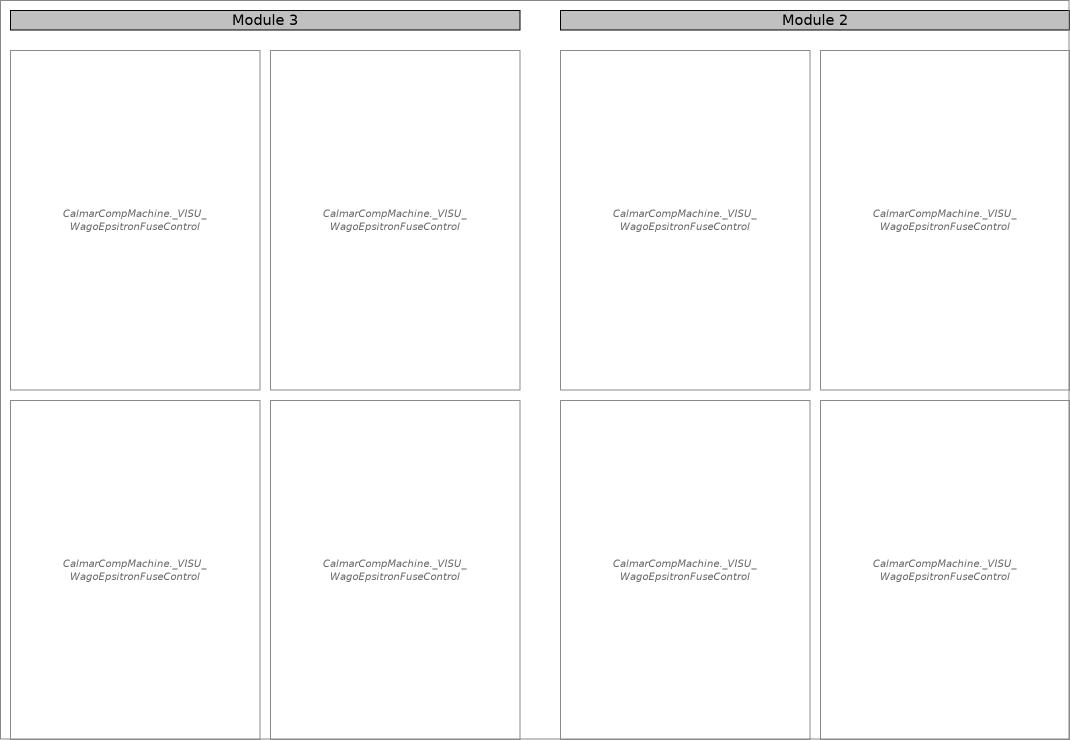
VISUALIZATION _VISU_FUSE_CONTROL  // 1070x740
VAR_IN_OUT
	mInst : FB_WeuPowerControl;
END_VAR
    Frame (820,50 250x340)
        shows CalmarCompMachine._VISU_WagoEpsitronFuseControl(m_Inst_Fb := PRG_MACHINE.fbPowerControl.fb_EpsitronFuseControlF70M1)
    Frame (560,50 250x340)
        shows CalmarCompMachine._VISU_WagoEpsitronFuseControl(m_Inst_Fb := PRG_MACHINE.fbPowerControl.fb_EpsitronFuseControlF90M1)
    Frame (270,50 250x340)
        shows CalmarCompMachine._VISU_WagoEpsitronFuseControl(m_Inst_Fb := PRG_MACHINE.fbPowerControl.fb_EpsitronFuseControlF70M2)
    Frame (10,50 250x340)
        shows CalmarCompMachine._VISU_WagoEpsitronFuseControl(m_Inst_Fb := PRG_MACHINE.fbPowerControl.fb_EpsitronFuseControlF90M2)
    Frame (270,400 250x340), invisible if: TRUE
        shows CalmarCompMachine._VISU_WagoEpsitronFuseControl(m_Inst_Fb := PRG_MACHINE.fbPowerControl.fb_EpsitronFuseControlF122M2)
    Frame (10,400 250x340), invisible if: TRUE
        shows CalmarCompMachine._VISU_WagoEpsitronFuseControl(m_Inst_Fb := PRG_MACHINE.fbPowerControl.fb_EpsitronFuseControlF160M2)
    Frame (820,400 250x340), invisible if: TRUE
        shows CalmarCompMachine._VISU_WagoEpsitronFuseControl(m_Inst_Fb := PRG_MACHINE.fbPowerControl.fb_EpsitronFuseControlF122M1)
    Frame (560,400 250x340), invisible if: TRUE
        shows CalmarCompMachine._VISU_WagoEpsitronFuseControl(m_Inst_Fb := PRG_MACHINE.fbPowerControl.fb_EpsitronFuseControlF160M1)
    Rectangle (10,10 510x20), "Module 3"
    Rectangle (560,10 510x20), "Module 2"
END_VISUALIZATION

(* stored: Version 1.1.0.1, ProductVersion 3.1.4024.11
   Visu _VISU_FUSE_CONTROL: Id {b3ce711f-ed21-4c2e-80a8-4f424f8625b4} *)
